{attribute 'GeneratedUsingTerminal: KL3351-0003'}
{attribute addProperty BoxType "KL3351-0003"}
{attribute addProperty Id "Channel_1AT %Q*Channel_0514A8FA0"}
{attribute addProperty CRC "3350770634"}
{attribute addProperty Size "0"}
TYPE KL_C7B8B3CA :
STRUCT
	{attribute addProperty Name "Channel_1"}
	Channel_1 : Channel_0514A8FA;
END_STRUCT
END_TYPE
